INTERFACE ITF_CANControl

METHOD M_GetMessage : BOOL
VAR_INPUT
END_VAR
END_METHOD

METHOD M_PushMessage : BOOL
VAR_INPUT
	messageSend : ST_TxRxMessage;
END_VAR
END_METHOD

END_INTERFACE

(* stored: Version 1.1.0.1, ProductVersion 3.1.4024.11
   Itf ITF_CANControl: Id {43a4a58d-7839-4761-abf2-57b0c488cde9}
   Method M_GetMessage: Id {a20ab3d6-fa25-46b5-b9fb-53657e8f0388}
   Method M_PushMessage: Id {b6a2bd18-9b57-4d5d-a38d-f1640078abf6} *)
